Staubli VAL3: CALL.dtx

num nLoad[20]
string listCall = "_placePrinter"
public string sItems
string sCallTemp = "Disk://..//templates/call"
bool bInit
bool bMutex
